FUNCTION_BLOCK SUBSCRIBE_24 (* Subscribe to a PUBLISH_24 Block *)
  (* Description: Copyright (c) 2017 fortiss GmbH This program and the accompanying materials are made available under the terms of the Eclipse Public License 2.0 which is available at https://www.eclipse.org/legal/epl-2.0/ SPDX-License-Identifier: EPL-2.0 *)
  (* Version 3.0, 2025-04-14, Patrick Aigner, changed package *)
  (* Version 1.0, 2017-10-25, Alois Zoitl, fortiss GmbH, initial API and implementation and/or initial documentation *)
  PACKAGE iec61499::net;
  {SET_ATTRIBUTE(eclipse4diac::core::GenericClassName, 'GEN_SUBSCRIBE')}
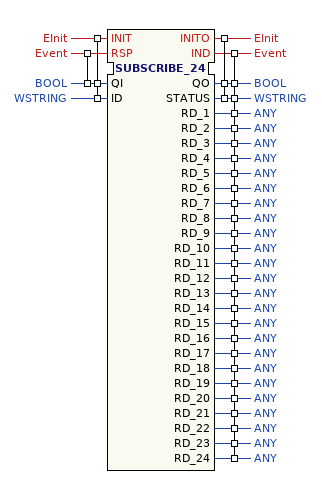
  EVENT_INPUT
    INIT : EInit WITH QI, ID;
    RSP WITH QI;
  END_EVENT
  EVENT_OUTPUT
    INITO : EInit WITH QO, STATUS;
    IND WITH QO, STATUS, RD_1, RD_2, RD_3, RD_4, RD_5, RD_6, RD_7, RD_8, RD_9, RD_10, RD_11, RD_12, RD_13, RD_14, RD_15, RD_16, RD_17, RD_18, RD_19, RD_20, RD_21, RD_22, RD_23, RD_24; (* New data available *)
  END_EVENT
  VAR_INPUT
    QI : BOOL;
    ID : WSTRING;
  END_VAR
  VAR_OUTPUT
    QO : BOOL;
    STATUS : WSTRING;
    RD_1 : ANY;
    RD_2 : ANY;
    RD_3 : ANY;
    RD_4 : ANY;
    RD_5 : ANY;
    RD_6 : ANY;
    RD_7 : ANY;
    RD_8 : ANY;
    RD_9 : ANY;
    RD_10 : ANY;
    RD_11 : ANY;
    RD_12 : ANY;
    RD_13 : ANY;
    RD_14 : ANY;
    RD_15 : ANY;
    RD_16 : ANY;
    RD_17 : ANY;
    RD_18 : ANY;
    RD_19 : ANY;
    RD_20 : ANY;
    RD_21 : ANY;
    RD_22 : ANY;
    RD_23 : ANY;
    RD_24 : ANY;
  END_VAR
  (* Service APPLICATION/RESOURCE: Subscribe to a PUBLISH_24 Block *)
END_FUNCTION_BLOCK
